// TIA Portal V16 export
// export: Created 2021-11-12T13:32:45.057222Z, ExportSetting WithDefaults, DisplayName Totally Integrated Automation Portal, DisplayVersion V16 Update 3, DisplayName TIA Portal Version Control Interface, DisplayVersion V16 Update 2, DisplayName TIA Portal Openness, DisplayVersion V16 Update 3, DisplayName SINAMICS Startdrive Advanced, DisplayVersion V16 Update 5, DisplayName SINAMICS Startdrive G130, G150, S120, S150, SINAMICS MV, S210, DisplayVersion V16 Update 5, DisplayName SINAMICS Startdrive G110M, G120, G120C, G120D, G120P, G115D, DisplayVersion V16 Update 5, DisplayName STEP 7 Professional, DisplayVersion V16 Update 3, DisplayName STEP 7 Safety, DisplayVersion V16, DisplayName WinCC UA Professional, DisplayVersion V16 Update 3
DATA_BLOCK "HMI_PARAM_BSN3"   // DB144
{ S7_Optimized_Access := 'TRUE' }
VERSION : 0.1
// stored: AutoNumber true, DBAccessibleFromOPCUA true, IsOnlyStoredInLoadMemory false, IsRetainMemResEnabled false, IsWriteProtectedInAS false, MemoryReserve 100
   VAR
      xxxxx___BinarySensors___xxxxx : Byte;
      xxxxx___BinaryOthers___xxxxx : Byte;
      xxxxx___AnalogueSensors___xxxxx : Byte;
      xxxxx___Drives___xxxxx : Byte;
      xxxxx___Others___xxxxx : Byte;
      PartCounter { S7_SetPoint := 'True'} : "UDT_PartCounter_Parameter";
      CL01 : "UDT_PartCounter_Parameter";
      xxxxx___SensorAlarms___xxxxx : Byte;
      Furnace : "UDT_DI_Mon_Parameter";   // from furnace
      LiveBit : "UDT_DI_Mon_Parameter";   // communication
      DataTracking : "UDT_DI_Mon_Parameter";   // part on senzor is not in data tracking
      Senzor : "UDT_DI_Mon_Parameter";   // part in data tracking is not on senzor
      Alarm_5 : "UDT_DI_Mon_Parameter";
      Alarm_6 : "UDT_DI_Mon_Parameter";
      Alarm_7 : "UDT_DI_Mon_Parameter";
      Alarm_8 : "UDT_DI_Mon_Parameter";
      Alarm_9 : "UDT_DI_Mon_Parameter";
      ES { S7_SetPoint := 'True'} : "UDT_DI_Mon_Parameter";   // E-stop
      xxxxx___ProcessAlarms___xxxxx : Byte;
      CL2 : "UDT_DI_Mon_Parameter";   // Box full alarm
      CL01_Warn : "UDT_DI_Mon_Parameter";   // Box full warning
   END_VAR
BEGIN
   CL01_Warn.Func := 16#2;
END_DATA_BLOCK
